(* PLC project Unnamed, Unknown Unnamed 1 *)
(* stored: creationDateTime 2023-03-10T10:37:17, modificationDateTime 2023-03-15T15:56:42 *)

(* ISBN: 978-3-8085-3450-2, Aufgabe 4 *)
FUNCTION_BLOCK Smoke_Detection_System
  VAR_INPUT
    IN1 : BOOL;
    IN2 : BOOL;
    IN3 : BOOL;
    IN4 : BOOL;
  END_VAR
  VAR_OUTPUT
    OUT1 : BOOL;
    OUT2 : BOOL;
    OUT3 : BOOL;
  END_VAR

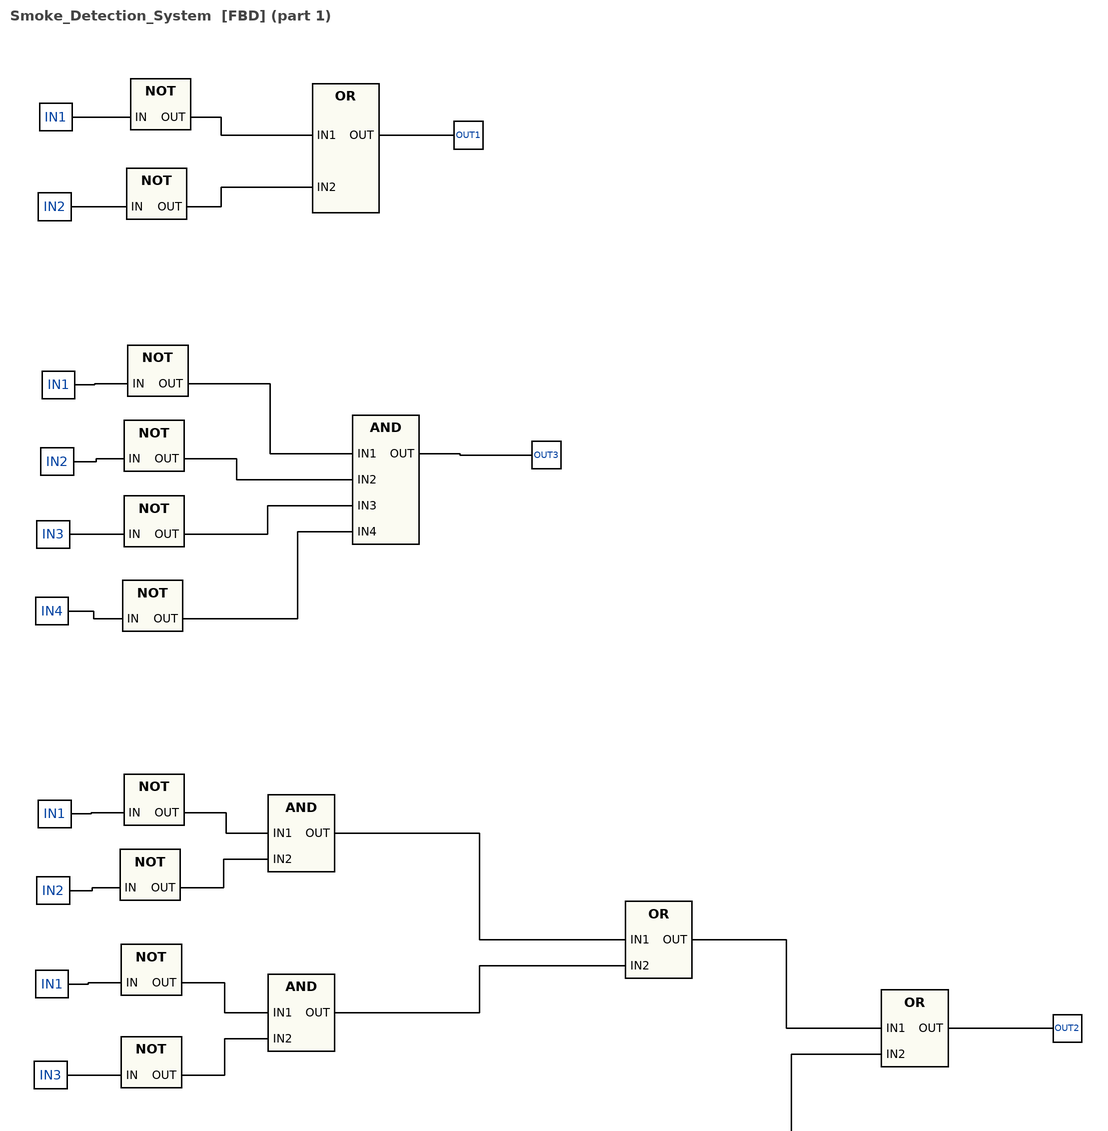
(* FBD diagram, written out as Structured Text *)
OUT1 := NOT IN1 OR NOT IN2;
OUT3 := NOT IN1 AND NOT IN2 AND NOT IN3 AND NOT IN4;
OUT2 := NOT IN1 AND NOT IN2 OR NOT IN1 AND NOT IN3 OR NOT IN1 AND NOT IN4 AND NOT IN3 AND NOT IN2 AND NOT IN2 AND NOT IN4 AND NOT IN3 AND NOT IN4;
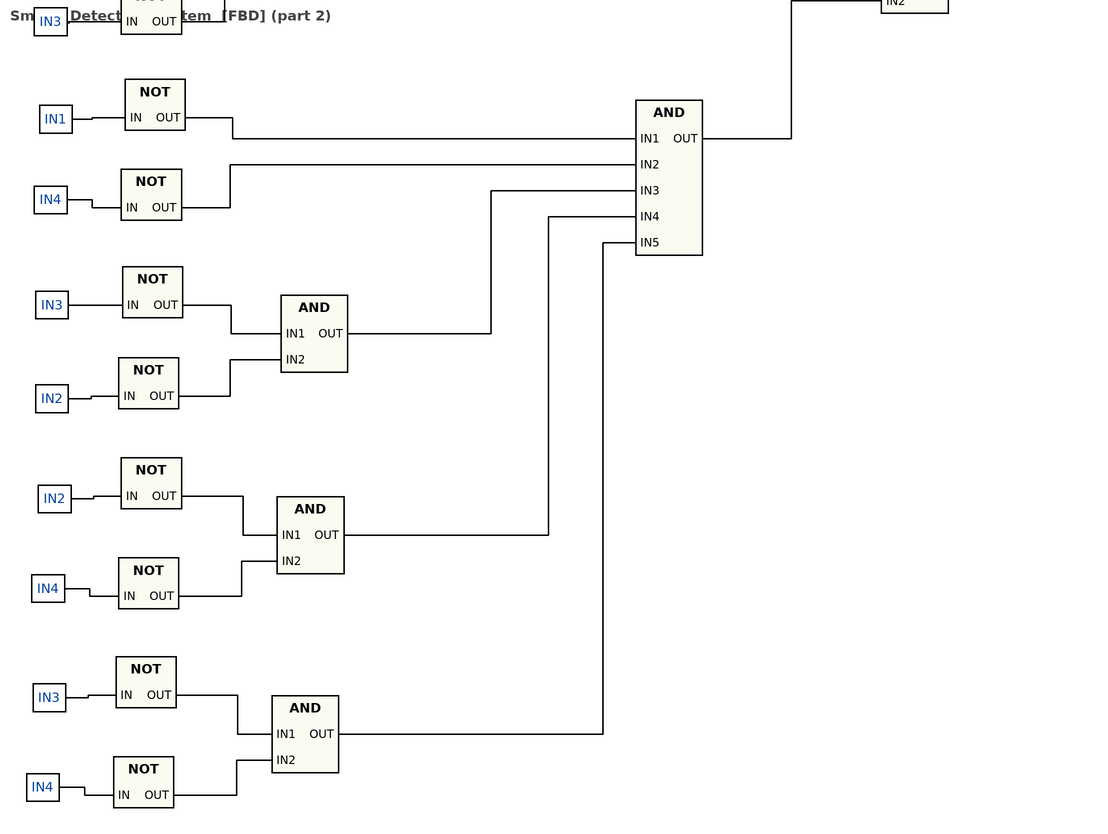
END_FUNCTION_BLOCK

CONFIGURATION config
  RESOURCE resource1 ON PLC
  END_RESOURCE
END_CONFIGURATION
